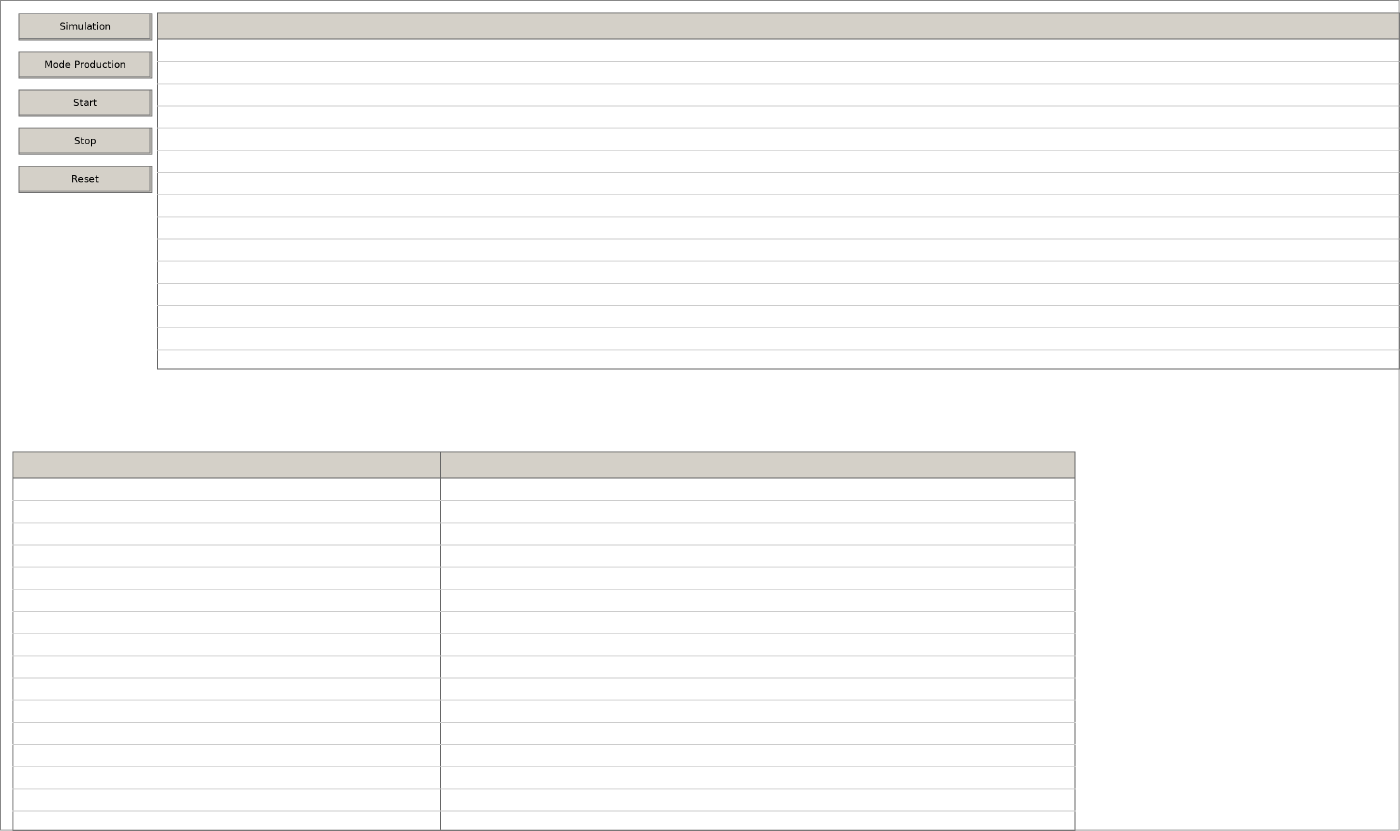
VISUALIZATION Vis_Machine  // 1577x937
    Button (21,15 150x30), "Simulation", colour toggle: GVL.g_bCmdSimulationOn, pressed state: g_bSimulationOn
        OnMouseClick: toggle GVL.g_bCmdSimulationOn
    Button (21,58 150x30), "Mode Production"
        OnMouseClick: execute { GVL_Area100.g_fbHmiMachCtrlsManager.q_eReqMode := E_PackML_Mode.Production; }
    Button (21,101 150x30), "Start", colour toggle: GVL_Area100.g_fbMachCtrlsManager.s_fbDiBtnStart[1].I_bIn
        OnMouseDown: execute { GVL_Area100.g_fbMachCtrlsManager.s_fbDiBtnStart[1].I_bIn := TRUE; }
        OnMouseUp: execute { GVL_Area100.g_fbMachCtrlsManager.s_fbDiBtnStart[1].I_bIn := FALSE; }
    Button (21,144 150x30), "Stop", colour toggle: GVL_Area100.g_fbMachCtrlsManager.s_fbDiBtnStop[1].I_bIn
        OnMouseDown: execute { GVL_Area100.g_fbMachCtrlsManager.s_fbDiBtnStop[1].I_bIn := TRUE; }
        OnMouseUp: execute { GVL_Area100.g_fbMachCtrlsManager.s_fbDiBtnStop[1].I_bIn := FALSE; }
    Button (21,187 150x30), "Reset", colour toggle: GVL_Area100.g_fbAlarmManager.s_bCmdResetFromDebug
        OnMouseDown: execute { GVL_Area100.g_fbAlarmManager.s_bCmdResetFromDebug := TRUE; }
        OnMouseUp: execute { GVL_Area100.g_fbAlarmManager.s_bCmdResetFromDebug := FALSE; }
    Group (14,509 1197x428)
        Table (482,0 715x428), data array: GVL_Area100.g_fbPackMLstatusManager.q_astPackML_status
            p3854506369: GVL_Area100.g_fbPackMLstatusManager.q_astPackML_status[INDEX].bAlwStateChange
            p1892666644: GVL_Area100.g_fbPackMLstatusManager.q_astPackML_status[INDEX].eActMode
            p338671338: GVL_Area100.g_fbPackMLstatusManager.q_astPackML_status[INDEX].eReqMode
            p2170511999: GVL_Area100.g_fbPackMLstatusManager.q_astPackML_status[INDEX].bModeChangeInProcess
            p3723444502: GVL_Area100.g_fbPackMLstatusManager.q_astPackML_status[INDEX].eActState
            p1218418051: GVL_Area100.g_fbPackMLstatusManager.q_astPackML_status[INDEX].eReqState
            p746581629: GVL_Area100.g_fbPackMLstatusManager.q_astPackML_status[INDEX].bStateEntry
            p3104783080: GVL_Area100.g_fbPackMLstatusManager.q_astPackML_status[INDEX].bStateChangeInProcess
            p2501879983: GVL_Area100.g_fbPackMLstatusManager.q_astPackML_status[INDEX].bStateComplete
            p7306298: GVL_Area100.g_fbPackMLstatusManager.q_astPackML_status[INDEX].bStateError
            p1933151965: GVL_Area100.g_fbPackMLstatusManager.q_astPackML_status[INDEX].tmStateTime
            p3863566920: GVL_Area100.g_fbPackMLstatusManager.q_astPackML_status[INDEX].nActSubState
            p2192122294: GVL_Area100.g_fbPackMLstatusManager.q_astPackML_status[INDEX].nReqSubState
            p400160035: GVL_Area100.g_fbPackMLstatusManager.q_astPackML_status[INDEX].bSubStateEntry
            p1128707560: Param_packML.c_nMaxModuleIndex
        Table (0,0 482x428), data array: GVL_Area100.g_fbPackMLstatusManager.q_asPackML_InstancePath
            p1128707560: Param_packML.c_nMaxModuleIndex
            p3854506369: GVL_Area100.g_fbPackMLstatusManager.q_asPackML_InstancePath[INDEX]
            p2232123230: PackML Instance Path
    Table (177,14 1400x402), data array: GVL_Area100.g_fbAlarmManager.q_astList
        p1128707560: Param_Alarms.c_nMaxNrOfListEntries
        p3854506369: GVL_Area100.g_fbAlarmManager.q_astList[INDEX].sInstancePath
        p1892666644: GVL_Area100.g_fbAlarmManager.q_astList[INDEX].nCfgIDnr
        p338671338: GVL_Area100.g_fbAlarmManager.q_astList[INDEX].nActivationTime
        p2170511999: GVL_Area100.g_fbAlarmManager.q_astList[INDEX].eCfgSeverity
        p3723444502: GVL_Area100.g_fbAlarmManager.q_astList[INDEX].eCfgAction
        p1218418051: GVL_Area100.g_fbAlarmManager.q_astList[INDEX].bStaResettable
        p746581629: GVL_Area100.g_fbAlarmManager.q_astList[INDEX].itfAlarmHandler
END_VISUALIZATION

(* stored: Version 1.1.0.1, ProductVersion 3.1.4024.12
   Visu Vis_Machine: Id {1cfdf8a3-835d-4fd5-988c-97981ccbbb80} *)
